Staubli VAL3: Day10.pjx

--- Day10.pjx ---
Parameters version=s8.13.1Cs9_BS2800 stackSize=5000 millimeterUnit=true
Program file=calc_score.pgx
Program file=start.pgx
Program file=stop.pgx
Data file=Day10.dtx
Library alias=util path=Disk://helpers/helpers.pjx
Library alias=math path=Disk://math/math.pjx
Library alias=str path=Disk://string/string.pjx
Library alias=stat path=Disk://statistics/statistics.pjx
Type name=lists path=Disk://types/lists/lists.pjx

--- Day10.dtx ---
string sInput
lists lResult
  [0]
    string sString
string sQueue
string sCorrupt
num nSum
num nCompletion
bool bCorrupt
num nResult

--- start.pgx ---
program start()
  local num l_nElement
  local num l_nResult
  local num l_nBracket
begin

  // read file
  call util:readFile("Disk://input_day10.txt", sInput)
  // sInput[0] = "[({(<((...."

  call str:splitString(sInput,"", lResult)
  // lResult.sString[0] = "["
  // lResult.sString[1] = "("

  // PUZZLE 1
  l_nResult = 0
  resize(sCorrupt,1,1)
  sCorrupt = ""

  for l_nElement = 0 to size(lResult)-1
    // reset sQueue
    resize(sQueue,1,1)
    sQueue = ""
    for l_nBracket = 0 to size(lResult[l_nElement].sString)-1
      if lResult[l_nElement].sString[l_nBracket] == "(" or lResult[l_nElement].sString[l_nBracket] == "<" or lResult[l_nElement].sString[l_nBracket] == "[" or lResult[l_nElement].sString[l_nBracket] == "{"
        append(sQueue)
        sQueue[size(sQueue)-1] = lResult[l_nElement].sString[l_nBracket]
      elseIf lResult[l_nElement].sString[l_nBracket] == ")" or lResult[l_nElement].sString[l_nBracket] == ">" or lResult[l_nElement].sString[l_nBracket] == "]" or lResult[l_nElement].sString[l_nBracket] == "}"
        if(sQueue[size(sQueue)-1] == "(" and lResult[l_nElement].sString[l_nBracket] == ")") or (sQueue[size(sQueue)-1] == "<" and lResult[l_nElement].sString[l_nBracket] == ">") or (sQueue[size(sQueue)-1] == "[" and lResult[l_nElement].sString[l_nBracket] == "]") or (sQueue[size(sQueue)-1] == "{" and lResult[l_nElement].sString[l_nBracket] == "}")
          delete(sQueue[size(sQueue)-1])
        else
          // Line corrupt!
          append(sCorrupt)
          sCorrupt[size(sCorrupt)-2] = lResult[l_nElement].sString[l_nBracket]
          // break out of this for-loop
          l_nBracket = 1000
          //endIf
        endIf

      endIf
    endFor
  endFor

  delete(sCorrupt[size(sCorrupt)-1])

  // Calculate sum
  nSum = 0
  for l_nElement = 0 to size(sCorrupt)-1
    if sCorrupt[l_nElement] == ")"
      nSum = nSum + 3
    endIf
    if sCorrupt[l_nElement] == "]"
      nSum = nSum + 57
    endIf
    if sCorrupt[l_nElement] == "}"
      nSum = nSum + 1197
    endIf
    if sCorrupt[l_nElement] == ">"
      nSum = nSum + 25137
    endIf

  endFor

  ? "PUZZLE 1:"
  call util:printNum(nSum)
  ? "############"
  // 392043

  // PUZZLE 2
  nSum = 0

  for l_nElement = 0 to size(lResult)-1
    // reset sQueue
    bCorrupt = false
    resize(sQueue,1,1)
    sQueue = ""
    for l_nBracket = 0 to size(lResult[l_nElement].sString)-1
      if lResult[l_nElement].sString[l_nBracket] == "(" or lResult[l_nElement].sString[l_nBracket] == "<" or lResult[l_nElement].sString[l_nBracket] == "[" or lResult[l_nElement].sString[l_nBracket] == "{"
        append(sQueue)
        sQueue[size(sQueue)-1] = lResult[l_nElement].sString[l_nBracket]
      elseIf lResult[l_nElement].sString[l_nBracket] == ")" or lResult[l_nElement].sString[l_nBracket] == ">" or lResult[l_nElement].sString[l_nBracket] == "]" or lResult[l_nElement].sString[l_nBracket] == "}"
        if(sQueue[size(sQueue)-1] == "(" and lResult[l_nElement].sString[l_nBracket] == ")") or (sQueue[size(sQueue)-1] == "<" and lResult[l_nElement].sString[l_nBracket] == ">") or (sQueue[size(sQueue)-1] == "[" and lResult[l_nElement].sString[l_nBracket] == "]") or (sQueue[size(sQueue)-1] == "{" and lResult[l_nElement].sString[l_nBracket] == "}")
          delete(sQueue[size(sQueue)-1])
          bCorrupt = false
        else
          // Line not complete!
          // break out of this for-loop
          bCorrupt = true
          l_nBracket = 1000
        endIf
      endIf
    endFor
    if bCorrupt == false
      call calc_score()
    endIf
  endFor

  delete(nCompletion[size(sCorrupt)])

  call stat:getMedian(nCompletion, nResult)
  ? "PUZZLE 2:"
  call util:printNum(nResult)


end

--- calc_score.pgx ---
program calc_score()
  local num l_nElement
begin

  append(nCompletion)

  for l_nElement = (size(sQueue)-1) to 0 step -1

    if sQueue[l_nElement] == "("
      nCompletion[size(nCompletion)-2] = 5*nCompletion[size(nCompletion)-2] + 1
    endIf
    if sQueue[l_nElement] == "["
      nCompletion[size(nCompletion)-2] = 5*nCompletion[size(nCompletion)-2] + 2
    endIf
    if sQueue[l_nElement] == "{"
      nCompletion[size(nCompletion)-2] = 5*nCompletion[size(nCompletion)-2] + 3
    endIf
    if sQueue[l_nElement] == "<"
      nCompletion[size(nCompletion)-2] = 5*nCompletion[size(nCompletion)-2] + 4
    endIf

  endFor


end
